FUNCTION F_CheckDivDint : DINT
VAR_INPUT
	divisor: DINT;
END_VAR

IF divisor = 0 THEN
	F_CheckDivDint:=1;
ELSE
	F_CheckDivDint:=divisor;
END_IF;

END_FUNCTION

(* stored: Version 1.1.0.1, ProductVersion 3.1.4022.6
   POU F_CheckDivDint: Id {68d52b2e-ba9e-4714-8d3b-214a99ccafab}, SpecialFunc None *)
